(* IEC 61131-3 sources: Lasal/CPU_5344_V01/Class/ValuePlusOffset, 1 file *)

(* ---- ValuePlusOffset.st ---- *)
(*!
<Class
	Name               = "ValuePlusOffset"
	Revision           = "0.0"
	RealtimeTask       = "true"
	DefRealtime        = "2 ms"
	CyclicTask         = "false"
	BackgroundTask     = "false"
	Sigmatek           = "false"
	OSInterface        = "false"
	HighPriority       = "false"
	Automatic          = "false"
	UpdateMode         = "Prescan"
	SharedCommandTable = "true"
	Objectsize         = "(284,120)">
	<Channels>
		<Server Name="ClassSvr" Visualized="false" Initialize="false" WriteProtected="true" Retentive="false"/>
		<Server Name="Offset" Visualized="true" Initialize="false" WriteProtected="false" Retentive="SRam"/>
		<Client Name="iEncoder" Required="true" Internal="false"/>
	</Channels>
</Class>
*)
ValuePlusOffset : CLASS
  //Servers:
	ClassSvr 	: SvrChCmd_DINT;
	Offset 	: SvrCh_DINT;
  //Clients:
	iEncoder 	: CltCh_DINT;
  //Variables:
  //Functions:

	FUNCTION VIRTUAL GLOBAL RtWork
		VAR_INPUT
			EAX 	: UDINT;
		END_VAR
		VAR_OUTPUT
			state (EAX) 	: UDINT;
		END_VAR;

	FUNCTION VIRTUAL GLOBAL ClassSvr::Read
		VAR_OUTPUT
			output (EAX) 	: DINT;
		END_VAR;
  //Tables:
	FUNCTION @STD
		VAR_OUTPUT
			ret_code	: CONFSTATES;
		END_VAR;
	FUNCTION GLOBAL TAB @CT_;
END_CLASS;

FUNCTION VIRTUAL GLOBAL ValuePlusOffset::ClassSvr::Read
	VAR_OUTPUT
		output (EAX) 	: DINT;
	END_VAR
    ClassSvr := iEncoder.Read() + Offset;

	output := ClassSvr;

END_FUNCTION

FUNCTION VIRTUAL GLOBAL ValuePlusOffset::RtWork
	VAR_INPUT
		EAX 	: UDINT;
	END_VAR
	VAR_OUTPUT
		state (EAX) 	: UDINT;
	END_VAR
    ClassSvr := iEncoder.Read() + Offset;

	state := READY;

END_FUNCTION
